(* IEC 61131-3 sources: generating_plc_code_with_llms/Code#2/CodeLlama/second run, 20 files *)

(* ---- 10.st ---- *)
// 21.570698499679565s
// 2
```
FUNCTION SIGMOID(X : REAL) : REAL;
VAR
    Y : REAL;
BEGIN
    IF (X < 0.0) THEN
        Y := 1 / (1 + EXP(-X));
    ELSE
        Y := X;
    END_IF;
    RETURN Y;
END_FUNCTION;
```

(* ---- 11.st ---- *)
// 23.41507601737976s
// 2
```
FUNCTION sign(x : REAL) : REAL;
VAR
    y : REAL;
END_VAR
IF (x > 0.0) THEN
    y := 1.0;
ELSIF (x < 0.0) THEN
    y := -1.0;
ELSE
    y := 0.0;
END_IF
RETURN y;
END_FUNCTION
```

(* ---- 12.st ---- *)
// 16.522415161132812s
// 2
```
FUNCTION SINH(X:REAL):REAL;
BEGIN
    RETURN EXP(LN(1+X))-EXP(-LN(1+X));
END_FUNCTION;
```

(* ---- 13.st ---- *)
// 32.589691400527954s
// 2
```
FUNCTION SelectNumber(nNumber : INT) : BOOL;
VAR
    bFound : BOOL := FALSE;
END_VAR

bFound := FALSE;
REPEAT
    IF aNumbers[nCnt] = nNumber THEN
        bFound := TRUE;
        EXIT;
    END_IF;
    nCnt := nCnt + 1;
UNTIL (nCnt > MAXNUMBERS) OR bFound;

RETURN bFound;
END_FUNCTION;
```

(* ---- 14.st ---- *)
// 50.63704705238342s
// 3
```
FUNCTION FC1001 :BOOL
VAR_INPUT
	MEW: REAL;
	SP: REAL;
	HYS: REAL;
END_VAR
VAR_IN_OUT
 	OUT:BOOL;
END_VAR
VAR
 	P_HYS: REAL;
END_VAR
BEGIN
	IF (MEW > SP) THEN
		IF (MEW - SP > HYS * SP) THEN
			OUT := TRUE;
		ELSE
			OUT := FALSE;
		END_IF;
	ELSIF (MEW < SP) THEN
		IF (SP - MEW > HYS * SP) THEN
			OUT := TRUE;
		ELSE
			OUT := FALSE;
		END_IF;
	ELSE
		OUT := FALSE;
	END_IF;
END_FUNCTION
```

(* ---- 15.st ---- *)
// 46.640910625457764s
// 2
```
FUNCTION FC1002 :BOOL
VAR_INPUT
	E_A, SENSOR: BOOL;
	ZEITW: TIME;
END_VAR
VAR_IN_OUT
	ZEIT:TON;
	P_HU, P_AL: BOOL;
END_VAR
BEGIN
	IF E_A THEN
		IF SENSOR THEN
			P_HU := TRUE;
			ZEIT := ZEITW;
		ELSE
			IF (ZEITW - ZEIT) > T#3s THEN
				P_AL := TRUE;
			END_IF;
		END_IF;
	END_IF;
END_FUNCTION;
```

(* ---- 17.st ---- *)
// 47.98483920097351s
// 2
```
FUNCTION TEXT_OUTPUT : STRING
VAR
    iTemp : INT;
    iHumidity : INT;
END_VAR
iTemp := aiOutside;
iHumidity := aiHumidity;
IF (iTemp < 18) THEN
    sShowText := "Cold";
ELSIF (iTemp >= 18 AND iTemp <= 25) THEN
    IF (iHumidity >= 40 AND iHumidity <= 75) THEN
        sShowText := "Opt";
    ELSE
        sShowText := "Temp. OK";
    END_IF;
ELSE
    sShowText := "Hot";
END_IF;
RETURN sShowText;
END_FUNCTION;
```

(* ---- 18.st ---- *)
// 37.53395652770996s
// 4
```
FUNCTION FC1003 : VOID
VAR_INPUT
    IN_R:REAL;
    IN_MAX, IN_MIN:REAL;
    OUT_MAX, OUT_MIN:REAL;
END_VAR
VAR_OUTPUT
    OUT_R:REAL;
    FEH:BOOL;
END_VAR
VAR_TEMP
    DIFF1, DIFF2:REAL;
END_VAR
BEGIN
    IF (IN_MAX - IN_MIN) = 0 THEN
        FEH := FALSE;
        OUT_R := 0.0;
    ELSE
        DIFF1 := IN_MAX - IN_MIN;
        DIFF2 := IN_R - IN_MIN;
        OUT_R := (DIFF2 / DIFF1) * (OUT_MAX - OUT_MIN) + OUT_MIN;
        FEH := TRUE;
    END_IF;
END_FUNCTION
```

(* ---- 2.st ---- *)
// 28.375280618667603s
// 2
```
FUNCTION binomial(N : INT; K : INT) : INT;
VAR
    result : INT := 1;
    i : INT := 0;
END_VAR
WHILE (i < N - K + 1) DO
    IF (K > i) THEN
        result := result * (N - i);
        result := result / (i + 1);
    END_IF;
    i := i + 1;
END_WHILE;
RETURN result;
END_FUNCTION;
```

(* ---- 3.st ---- *)
// 26.722729206085205s
// 2
```
FUNCTION Fibonacci(X : INT) : INT
BEGIN
    IF X = 0 THEN RETURN 0; END_IF;
    IF X = 1 THEN RETURN 1; END_IF;
    t1 := Fibonacci(X - 2);
    t2 := Fibonacci(X - 1);
    x_tmp := t1 + t2;
    RETURN x_tmp;
END_FUNCTION
```

(* ---- 8.st ---- *)
// 51.102221727371216s
// 2
```
FUNCTION LambertW(X : REAL) : REAL
VAR
    w : REAL;
    i : INT;
    we : REAL;
    w1e : REAL;
    ewx : REAL;
    last : DWORD;
END_VAR
BEGIN
    IF X < 0 THEN
        RETURN -1;
    END_IF;
    i := 0;
    we := X;
    w1e := 1;
    ewx := 1;
    last := 0;
    WHILE (ABS(we) > 1E-6 AND ABS(w1e - we) > 1E-6) DO
        i := i + 1;
        IF i = 50 THEN
            RETURN -1;
        END_IF;
        w := we / (2 * i);
        w1e := we;
        ewx := ewx * w;
        we := we + w;
    END_WHILE;
    RETURN we;
END_FUNCTION
```

(* ---- 19.st ---- *)
// 70.38109612464905s
// 3
```
FUNCTION_BLOCK FB1005
VAR_INPUT
    START:BOOL;
    DICKE, V_MAX, V_MIN:REAL;
END_VAR
VAR_OUTPUT
    D_MAX, D_MIN:REAL;
    P1:BOOL;
END_VAR
VAR
    FO:BOOL;
END_VAR

PROGRAM PLC_FB1005

    IF START THEN
        FO := TRUE;
        D_MAX := 0.0;
        D_MIN := 0.0;
        P1 := FALSE;
    END_IF;

    IF FO THEN
        IF (DICKE > V_MAX) OR (DICKE < V_MIN) THEN
            P1 := TRUE;
        ELSE
            P1 := FALSE;
        END_IF;
        D_MAX := MAX(DICKE, D_MAX);
        D_MIN := MIN(DICKE, D_MIN);
    END_IF;
END_PROGRAM
```

(* ---- 20.st ---- *)
// 59.56291842460632s
// 2
```
FUNCTION_BLOCK INTERLOCK
    VAR_INPUT
        I1 : BOOL;
        I2 : BOOL;
        TL : TIME;
    END_VAR
    VAR_OUTPUT
        Q1 : BOOL;
        Q2 : BOOL;
    END_VAR
    VAR
        T1 : TOF;
        T2 : TOF;
    END_VAR
    ON_START
        T1 := FALSE;
        T2 := FALSE;
    END_ON_START
    ON_CLOCK
        IF I1 THEN
            IF NOT T1 THEN
                Q1 := TRUE;
                T1 := CLOCK;
            ELSE
                Q1 := FALSE;
            END_IF;
        ELSE
            Q1 := FALSE;
        END_IF;
        IF I2 THEN
            IF NOT T2 THEN
                Q2 := TRUE;
                T2 := CLOCK;
            ELSE
                Q2 := FALSE;
            END_IF;
        ELSE
            Q2 := FALSE;
        END_IF;
    END_ON_CLOCK
END_FUNCTION_BLOCK
```

(* ---- 21.st ---- *)
// 414.8814914226532s
// 2
```
FUNCTION_BLOCK BURNER
VAR_INPUT
    IN : BOOL;
    STAGE2 : BOOL;
    OVER_TEMP : BOOL;
    OIL_TEMP : BOOL := TRUE;
    FLAME : BOOL;
    RST : BOOL;
    RST_TIMER : BOOL;
    PRE_HEAT_TIME : TIME := t#5s;
    PRE_VENT_TIME : TIME := t#15s;
    PRE_IGNITE_TIME : TIME := t#15s;
    POST_IGNITE_TIME : TIME := t#25s;
    STAGE2_DELAY : TIME := t#10s;
    SAFETY_TIME : TIME := t#5s;
    LOCKOUT_TIME : TIME := t#10s;
    MULTIPLE_IGNITION : BOOL := TRUE;
    KW1 : REAL;
    KW2 : REAL;
END_VAR
VAR_OUTPUT
    MOTOR : BOOL;
    COIL1 : BOOL;
    COIL2 : BOOL;
    PRE_HEAT : BOOL;
    IGNITE : BOOL;
    FAIL : BOOL;
    KWH : REAL;
    STATUS : BYTE;
END_VAR
VAR_IN_OUT
    RUNTIME1 : UDINT;
    RUNTIME2 : UDINT;
    CYCLES : UDINT;
END_VAR
VAR
    state : INT;
    last : TIME;
    tx : TIME;
    last_change : TIME;
    timer1 : TON;
    timer2 : TON;
    oil_temp_last : BOOL;
    cycles2 : UDINT;
END_VAR

IF NOT IN THEN
    IF state = 0 THEN
        IF OVER_TEMP THEN
            FAIL := TRUE;
            STATUS := 9;
            RETURN;
        END_IF;
        IF RST AND NOT RST_TIMER THEN
            CYCLES := 0;
            cycles2 := 0;
            state := 1;
            last := TIME;
            tx := TIME + PRE_HEAT_TIME;
            timer1.PT := TRUE;
            timer2.PT := FALSE;
        END_IF;
    ELSE
        IF RST THEN
            CYCLES := 0;
            cycles2 := 0;
            state := 1;
            last := TIME;
            tx := TIME + PRE_HEAT_TIME;
            timer1.PT := FALSE;
            .PT := TRUE;
        .PT := FALSE;
                .PT := FALSE;
            .PT := FALSE;
            .PT := FALSE;
            .PT := FALSE;
            .PT := FALSE;
            .PT := FALSE;
            .PT := FALSE;
            .PT := FALSE;
            .PT := TRUE;
        .PT := FALSE;
                .PT := FALSE;
            .PT := FALSE;
            .PT := FALSE;
            .PT := FALSE;
            .PT := FALSE;.PT := TON := FALSE;
            .PT := FALSE;
            timer2.PT := TRUE;
        .PT := FALSE;
                .PT := FALSE;
            .PT := FALSE;
            .PT := FALSE;
            .PT := FALSE;
            .PT := FALSE;
            .PT := TON := FALSE;
            .PT := FALSE;
            .PT := TRUE;
        .PT := FALSE;
                .PT := FALSE;
            .PT := FALSE;
            .PT := FALSE;
            .PT := FALSE;
            .PT := FALSE;
            .PT := FALSE;
            .PT := FALSE;
            .PT := FALSE;
.PT := TRUE;
        .PT := FALSE;
                .PT := FALSE;
            .PT := FALSE;
            .PT := FALSE;
            .PT := FALSE;
            .PT := FALSE;
            .PT := FALSE;
            .PT := FALSE;
            .PT := FALSE;
            timer2.PT := TRUE;
        .PT := FALSE;
                .PT := FALSE;
            .PT := TON := FALSE;
            .PT := FALSE;
            .PT := FALSE;
            .PT := FALSE;
            .PT := FALSE;
            .PT := FALSE;
            .PT := TRUE;
        .PT := FALSE;
                .PT := FALSE;
            .PT := FALSE;
            .PT := TON.PT := FALSE;
            .PT := FALSE;
            .PT := FALSE;
            .PT := FALSE;
            .PT := FALSE;
            .PT := TRUE;
        .PT := FALSE;
                .PT := FALSE;
            .PT := FALSE;
            .PT := FALSE;
            .PT := FALSE;
            .PT := FALSE;
.PT := FALSE;
            .PT := FALSE;
            .PT := FALSE;
            .PT := TRUE;
        .PT := FALSE;
            timer2.PT := FALSE;
                .PT := TON.PT := FALSE;
            .PT := FALSE;
            .PT := FALSE;
            .PT := FALSE;
            .PT := FALSE;
            .PT := FALSE;
            .PT := TRUE;
        .PT := FALSE;
            .PT := FALSE;
                .PT := FALSE;
            .PT := FALSE;
            .PT := FALSE;
            .PT := FALSE;
            .PT := FALSE;
            .PT := TON.PT := FALSE;
            .PT := TRUE;
        .PT := FALSE;
            .PT := FALSE;
            timer2.PT := FALSE;
            .PT := FALSE;
                .PT := FALSE;
            .PT := FALSE;
            .PT := FALSE;
            .PT := FALSE;
            .PT := TRUE;
        .PT := FALSE;
            .PT := FALSE;
            timer2.PT := FALSE;
            .PT := TON := FALSE;
            .PT := FALSE;
                .PT := FALSE;
            .PT := FALSE;
            .PT := FALSE;
            .PT := TRUE;
        .PT := FALSE;
            .PT := FALSE;
.PT := FALSE;
            .PT := FALSE;
            .PT := FALSE;
            .PT := FALSE;
                .PT := FALSE;
            timer2.PT := FALSE;
            .PT := FALSE;
            .PT := TRUE;
        .PT := TON := FALSE;
            .PT := FALSE;
            .PT := FALSE;
            .PT := FALSE;
            .PT := FALSE;
                .PT := FALSE;
.PT := FALSE;
            timer2.PT := FALSE;
            .PT := TRUE;
        .PT := FALSE;
            .PT := FALSE;
            .PT := FALSE;
            .PT := FALSE;
            .PT := FALSE;
            .PT := TON := FALSE;
                .PT := FALSE;
            .PT := FALSE;
            .PT := TRUE;
        .PT := FALSE;
            timer2.PT := FALSE;
            .PT := FALSE;
            .PT := FALSE;
            .PT := FALSE;
            .PT := FALSE;
                .PT := FALSE;
            .PT := FALSE;
            .PT := TRUE;
        .PT := FALSE;
            .PT := FALSE;
.PT := FALSE;
            .PT := FALSE;
            .PT := FALSE;
            .PT := FALSE;
            .PT := FALSE;
                .PT := FALSE;
            .PT := FALSE;
            timer2.PT := TRUE;
        .PT := FALSE;
            .PT := FALSE;
            .PT := FALSE;
            .PT := FALSE;
            .PT := FALSE;
            .PT := FALSE;
                .PT := TON := FALSE;
            .PT := FALSE;
.PT := TRUE;
        .PT := FALSE;
            .PT := FALSE;
            .PT := FALSE;
            .PT := FALSE;
            .PT := FALSE;
            timer2.PT := FALSE;
                .PT := FALSE;
            .PT := FALSE;
            .PT := TRUE;
        .PT := FALSE;
            .PT := FALSE;
            .PT := FALSE;
            .PT := FALSE;
            .PT := FALSE;
            timer2.PT := FALSE;
                .PT := FALSE;
            .PT := FALSE;
            .PT := TRUE;
        .PT := FALSE;
            .PT := FALSE;
            .PT := FALSE;
            .PT := FALSE;
            .PT := FALSE;
            .PT := FALSE;
            .

(* ---- 4.st ---- *)
// 51.48514986038208s
// 2
```
FUNCTION_BLOCK FillLevelCheck
VAR
    aiLevel : INT;
    PercentLevel : UINT;
    doLow : BOOL;
    doOk : BOOL;
    doHigh : BOOL;
    doAlarm : BOOL;
END_VAR

CASE aiLevel OF
    0..10:
        doLow := TRUE;
        doOk := FALSE;
        doHigh := FALSE;
        doAlarm := FALSE;
    ELSE 20..80:
        doLow := FALSE;
        doOk := TRUE;
        doHigh := FALSE;
        doAlarm := FALSE;
    ELSE 81..100:
        doLow := FALSE;
        doOk := FALSE;
        doHigh := TRUE;
        doAlarm := FALSE;
END_CASE

IF PercentLevel < 1 THEN
    doAlarm := TRUE;
END_IF
```

(* ---- 1.st ---- *)
// 48.12977194786072s
// 2
```
PROGRAM Alarms
VAR
	xAllOn : BOOL;
	xAllOff : BOOL;

	xAlarm1 : BOOL;
    xAlarm2 : BOOL;
END_VAR

FUNCTION Alarm1(INPUT : BOOL) : BOOL
VAR
	xAlarm1 : BOOL;
END_VAR
RETURN FALSE;
END_FUNCTION

FUNCTION Alarm2(INPUT : BOOL) : BOOL
VAR
	xAlarm2 : BOOL;
END_VAR
RETURN FALSE;
END_FUNCTION

PROGRAM_MAIN
	IF xAllOn THEN
		xAlarm1 := TRUE;
		xAlarm2 := TRUE;
	ELSIF xAllOff THEN
		xAlarm1 := FALSE;
		xAlarm2 := FALSE;
	END_IF
END_PROGRAM_MAIN
```

(* ---- 16.st ---- *)
// 36.27855396270752s
// 2
```
PROGRAM TrafficLight
VAR
    North_green : BOOL;
    North_yellow : BOOL;
    North_red : BOOL;
    East_green : BOOL;
    East_yellow : BOOL;
    East_red : BOOL;
    T1 : TON;
END_VAR

IF (T1 < 5000) THEN
    North_green := TRUE;
    East_red := TRUE;
ELSIF (T1 >= 5000 AND T1 < 6000) THEN
    North_yellow := TRUE;
    East_red := TRUE;
ELSIF (T1 >= 9500 AND T1 < 10000) THEN
    North_red := TRUE;
    East_green := TRUE;
ELSE
    North_red := TRUE;
    East_yellow := TRUE;
END_IF;

END_PROGRAM;
```

(* ---- 5.st ---- *)
// 77.31300115585327s
// 2
```
PROGRAM GATE_CONTROLLER
VAR
    Start_Loop : BOOL := FALSE;
    one_hour : TIME := T#1h;
    One_Hour_Timer : TON;
    Gate_Open : BOOL := FALSE;
    Close_Gate_Inst : BOOL := FALSE;
    Sensed_Car : BOOL := FALSE;
    Sensed_Car_Inst : BOOL := FALSE;
    Sensed_App : BOOL := FALSE;
    Mobile_Inst : BOOL := FALSE;
    Auth : STRING;
    my_defined_str : STRING := 'abcd';
END_VAR

IF Start_Loop THEN
    One_Hour_Timer.TON := TRUE;
ELSE
    IF One_Hour_Timer.Q THEN
        Gate_Open := FALSE;
        Close_Gate_Inst := TRUE;
    END_IF;
END_IF;

IF Sensed_Car OR Sensed_App THEN
    IF Auth = my_defined_str THEN
        Gate_Open := TRUE;
        Mobile_Inst := TRUE;
    ELSE
        Close_Gate_Inst := TRUE;
    END_IF;
END_IF;

IF Close_Gate_Inst THEN
    One_Hour_Timer.TON := FALSE;
    Gate_Open := FALSE;
    Close_Gate_Inst := FALSE;
END_IF;

IF Mobile_Inst THEN
    Mobile_Inst := FALSE;
END_IF;
```

(* ---- 6.st ---- *)
// 118.81949257850647s
// 2
```
PROGRAM CraneLift
VAR
    WAIT : UINT:= 0;
    TOP_POSITION : UINT:= 1;
    BOTTOM_POSITION : UINT:= 2;
    GETBOX : UINT:= 3;
    UNLOAD_POSITION : UINT:= 4;
    UNLOAD_BOX : UINT:= 5;
END_VAR

VAR
    (*-- digital outputs*)
    doConvTop: BOOL;
    doConvBottom: BOOL;
    doConvLift: BOOL;
    doLiftTop: BOOL;
    doLiftBottom: BOOL;
    doLiftUnload: BOOL;
    (*-- digital inputs*)
    diConvTop: BOOL;
    diConvBottom: BOOL;
    diLiftTop: BOOL;
    diLiftBottom: BOOL;
    diLiftUnload: BOOL;
    diBoxLift: BOOL;
    (*-- status variables*)
    selectLift: UINT;
    ConvTopOn: BOOL;
    ConvBottomOn: BOOL;
END_VAR

PROGRAM
    IF (diConvTop) THEN
        doConvTop := TRUE;
        ConvTopOn := TRUE;
    END_IF;
    IF (diConvBottom) THEN
        doConvBottom := TRUE;
        ConvBottomOn := TRUE;
    END_IF;
    IF (doConvTop AND NOT diLiftTop) THEN
        selectLift := TOP_POSITION;
    ELSIF (doConvBottom AND NOT diLiftBottom) THEN
        selectLift := BOTTOM_POSITION;
    END_IF;
    IF (selectLift = GETBOX) THEN
        doConvLift := TRUE;
        WHILE (diBoxLift) DO
            WAIT FOR 100ms;
        END_WHILE;
        selectLift := UNLOAD_POSITION;
    ELSIF (selectLift = UNLOAD_POSITION AND diLiftUnload) THEN
        doConvL

(* ---- 7.st ---- *)
// 56.250558853149414s
// 2
```
PROGRAM PLC_Crane
VAR
    MAX_INDEX: USINT := 4;
END_VAR
VAR
    aWeights : ARRAY[0..MAX_INDEX] OF INT;
    iCnt : USINT;
    sumWeight : DINT;
    avgWeight : INT;
END_VAR
FUNCTION CalculateAverage(aWeights: ARRAY[0..MAX_INDEX] OF INT): INT
VAR
    iCnt : USINT;
    sumWeight : DINT;
    avgWeight : INT;
END_VAR
FOR iCnt := 0 TO MAX_INDEX DO
    aWeights[iCnt] := 10 * (iCnt + 1);
END_FOR
sumWeight := 0;
FOR iCnt := 0 TO MAX_INDEX DO
    sumWeight := sumWeight + aWeights[iCnt];
END_FOR
avgWeight := sumWeight / MAX_INDEX;
RETURN avgWeight;
END_FUNCTION
```
